FUNCTION TrackAndTraceInfo : STRING
VAR_INPUT
	stap : INT;	//Input parameter, huidige stap
END_VAR

CASE stap OF
	0:	TrackAndTraceInfo := 'Wachten op bestelling.';
	1:	TrackAndTraceInfo := 'Bestelling geplaatst!';
	2:	TrackAndTraceInfo := 'Bezorgen staat voor uw deur.';
	3:	TrackAndTraceInfo := 'Bestelling is in uw handen!';
	4:	TrackAndTraceInfo := 'Bestelling aanwezig bij ophaalpunt.';
	ELSE
		TrackAndTraceInfo := 'Status onbekend.';
END_CASE

END_FUNCTION

(* stored: Version 1.1.0.1, ProductVersion 3.1.4024.13
   POU TrackAndTraceInfo: Id {2ce61888-764b-4d6a-b722-76474068337d}, SpecialFunc None *)
